{attribute addProperty BoxType "EL6002-0000-0016"}
{attribute addProperty Id "StatusAT %I*Status_0CBEDEF8232.8751Data_InAT %I*ARRAY[0 ..21] OF USINT176220"}
{attribute addProperty CRC "186151800"}
{attribute addProperty SizeInBites "199"}
{attribute addProperty SizeInBytes "24.875"}
TYPE COM_Inputs_Channel_DABE08D3 :
STRUCT
	{attribute addProperty Name "Status"}
	Status AT %I* : Status_0CBEDEF8;
	{attribute addProperty Name "Data_In"}
	Data_In AT %I* : ARRAY[0 ..21] OF USINT;
END_STRUCT
END_TYPE

(* stored: Version 1.2.0.0, ProductVersion 3.1.4024.9
   DUT COM_Inputs_Channel_DABE08D3: Id {03231825-c7f0-4534-acc9-dbdcd75bc98e} *)
